{attribute 'pack_mode' := '1'}
TYPE TPearlingData :
STRUCT
		THead 	: ARRAY[PH_Left..PH_Right] OF TPearlingDataHead;
END_STRUCT
END_TYPE

(* stored: Version 1.1.0.1, ProductVersion 3.1.4022.12
   DUT TPearlingData: Id {3e71056a-c357-4e59-acec-29f9ff3cbba3} *)
